{attribute 'qualified_only'}
{attribute 'strict'}
TYPE E_PLCTPL_COMMAND :
(
	NONE	:= 0,
	
	RESET,
	INIT,
	STOP,
	ENABLE,
	DISABLE,
	OPEN,
	CLOSE
	
);
END_TYPE

(* stored: Version 1.1.0.1, ProductVersion 3.1.4022.16
   DUT E_PLCTPL_COMMAND: Id {384c1f9b-10c2-4511-9e8a-004d22171a66} *)
